{attribute 'pack_mode':='1'}
TYPE InboundToteParams :
STRUCT
	source_id : ModelIdentifier; // Identifier for the source inbound line.
	target_id : ModelIdentifier; // Identifier for the target work position.
END_STRUCT
END_TYPE

(* stored: Version 1.1.0.1, ProductVersion 3.1.4024.12
   DUT InboundToteParams: Id {5f5c34f5-9e70-40c7-8be2-6f505c24ea61} *)
